PROGRAM MAIN
VAR
END_VAR

END_PROGRAM

(* stored: Version 1.1.0.1
   POU MAIN: Id {9b8af115-f696-42b7-ba93-9f2918b47890} *)
